Fanuc KAREL source: ka00145.KL

-- PROVISIONAL review KL for V770-1; original PC SHA256 2ab32d2fd787c5135ba55a0bdb49d97704445109f32b0cd4556d2cee6f57cb4b
-- Incomplete behavior may be omitted. Consult companion uncertainty JSON. Do not deploy.
PROGRAM KA00145
%NOLOCKGROUP
-- UNRESOLVED_DECL SRC type=002010
-- UNRESOLVED_DECL DST type=002010
BEGIN
  -- UNRESOLVED_PC offsets 5-19; opcodes 22,22,1E
  -- UNRESOLVED_PC offsets 24-28; opcodes 7F
END KA00145
